PROGRAM OP90_CAMERA
VAR
END_VAR

OP90_LH_CMR_OK			:= TRUE;
OP90_RH_CMR_OK			:= TRUE;

END_PROGRAM

(* stored: Version 1.1.0.1, ProductVersion 3.1.4024.11
   POU OP90_CAMERA: Id {911a2e93-9e04-4a7f-9282-697f696d1304}, SpecialFunc None *)
